(**********************SISSI:Swap from Ink to Storage Flush*********************************)
FUNCTION_BLOCK FB_Auto_Cycles_Swap
VAR_INPUT
	Sensor1			:BOOL;
	Sensor4			:BOOL;
	Circ_Pump_L	:BOOL;
	Circ_Pump_R	:BOOL;
	Circ_normal_error:INT;
	btPurge			:BOOL;
	
END_VAR
VAR_OUTPUT
	state								:INT;
	error_code					:INT;
	
	SwapInfo						:INT;
	VacValve_V8					:BOOL;	//白墨负压阀
	PurValve_V7					:BOOL;//正压阀
	alternate_Pumping		:BOOL;//交替加墨
	Swapping_Done			:BOOL;
	Error					:BOOL;
END_VAR
VAR
	step						:INT;
	stepA,stepB1,	stepB2		:INT;
	Ton,ton7,ton10				:TON;
	
	FB_SQUARE					:FB_SQUARE;
	W,X,A,Z,Y:INT;
	cycle_r_trig1,cycle_r_trig2  :R_TRIG;      //循坏
	cycle_x1,cycle_x2				:INT;//循坏次数
	purge_F_trig:F_TRIG;
	dely_off_setoff:TON;
	dely_emstop:Tc2_Standard.TON;
	ton1:Tc2_Standard.TON;
END_VAR
VAR_IN_OUT
	initialize				:BOOL;
	swap					:BOOL;
	CYCLE					:INT;//"0:Cycle A: Swap white ink to storage ;1:Cycle B: Swap storage to white ink"
	setoff					:BOOL;
END_VAR

IF setoff OR GVL.Reset THEN 
	step:=99;
END_IF
CASE step OF 
0://waiting
	IF initialize THEN 
		step :=5;
	ELSIF swap THEN 
		step :=10;
	ELSIF setoff OR GVL.Reset THEN 
		step :=99;
	END_IF
	
(***********当状态=Idle时，错误代码等于循坏错误****************************************)
	IF  state=MUStateEnum.idle THEN 
		error_code:=Circ_normal_error;
	END_IF
(***********自复位****************************************)	
	ton1(IN:=Swapping_Done , PT:= T#1S, Q=> , ET=> );
	IF ton1.Q THEN 
		Swapping_Done:=FALSE;
	END_IF
5://OFF
	state:=MUStateEnum.off;
	error_code:=MUErrorEnum.no_error;
	stepA:=stepB1:=stepB2:=0;
	W:=X:=A:=Z:=Y:=0;
	SwapInfo:=SwapInfoEnum.NONE;
	dely_emstop(IN:=FALSE);

	VacValve_V8:=FALSE;
	PurValve_V7:=FALSE;	
	
	GVL.fill_W_in_swap_enable:=FALSE;
	GVL.fill_F_in_swap_enable:=FALSE;
	
		IF initialize THEN //idle,此状态，所有泵停止	
			initialize:=FALSE;
			state:=MUStateEnum.idle;					
			GVL.fill_W_in_swap_enable:=FALSE;
			step:=0;
		END_IF
10://idle,此状态，所有泵停止				
		IF swap THEN 
			swap:=FALSE;
			state:=MUStateEnum.swapping;
			error_code:=MUErrorEnum.no_error;
			step:=20;
		END_IF
		
		IF error_code<>0 THEN 			
			step:=100;
		END_IF

20://SWAPPING		
		IF CYCLE=0 THEN
			ACT_Cycle_A();			
		ELSIF CYCLE=1 THEN 
			ACT_Cycle_B1();	
		END_IF
		
		IF SwapInfo=SwapInfoEnum.AC_STORAGE_FLUSH_FINISHED OR 
			SwapInfo=SwapInfoEnum.AC_WHITE_INK_FINISHED THEN 
			stepA:=stepB1:=stepB2:=0;		
			Swapping_Done:=TRUE;
			state:=MUStateEnum.idle;
			step:=0;
		END_IF
99://setoff
	setoff :=FALSE;
	error:=FALSE;
	state:=MUStateEnum.off;
	error_code:=MUErrorEnum.no_error;
	stepA:=stepB1:=stepB2:=0;
	W:=X:=A:=Z:=Y:=0;
	SwapInfo:=SwapInfoEnum.NONE;
	dely_emstop(IN:=FALSE);
	VacValve_V8:=FALSE;
	PurValve_V7:=FALSE;	
	
	GVL.fill_W_in_swap_enable:=FALSE;
	GVL.fill_F_in_swap_enable:=FALSE;
	step:=0;
100://error
		error:=TRUE;
		state:=MUStateEnum.error;
		stepA:=stepB1:=stepB2:=0;
		W:=X:=A:=Z:=Y:=0;
		dely_emstop(IN:=FALSE);
		VacValve_V8:=FALSE;
		PurValve_V7:=FALSE;	
		
		GVL.fill_W_in_swap_enable:=FALSE;
		GVL.fill_F_in_swap_enable:=FALSE;		
		step:=0;
END_CASE

IF setoff OR GVL.Reset THEN 
	step:=99;
END_IF

dely_off_setoff(IN:=setoff , PT:=T#1S , Q=> , ET=> );
IF dely_off_setoff.Q THEN
	setoff:=FALSE;
END_IF

IF state<>MUStateEnum.off AND state<>MUStateEnum.error  THEN 
	IF GVL.Emstop_Button THEN 
		error:=TRUE;
		error_code:=MUErrorEnum.emergency_error;
		PurValve_V7:=FALSE;
		dely_emstop(IN:=TRUE , PT:=T#1S , Q=> , ET=> );
		IF dely_emstop.Q THEN 
			VacValve_V8:=FALSE;
			step:=100;
		END_IF
	END_IF
END_IF

ACTION ACT_Cycle_A:
(***************Swap from White Ink to Storage Flush*******************************************)
CASE StepA OF
0:
	SwapInfo:=SwapInfoEnum.AC_STORAGE_FLUSH_RUNS;
	Ton(IN:=FALSE );	
	VacValve_V8:=FALSE;
	PurValve_V7 :=FALSE;
	stepA:=10;
10://SET "Vac White" OFF (valve 8 ON) 
	//START Pressure Purge Time = T1 (valve 7 ON)
	VacValve_V8:=TRUE;
	PurValve_V7 :=TRUE;
	Ton(IN:=TRUE , PT:=LREAL_TO_TIME(T[1]*1000) , Q=> , ET=> );
	IF Ton.Q THEN 
		Ton(IN:=FALSE );	
		stepA:=20;
	END_IF
20://STOP Pressure purge (normal filling conditions) (valve 7 OFF)	
	PurValve_V7:=FALSE;
	stepA:=30;
30://START Sol. filling (alternating pump time: T2=ON, T3=OFF)
	//WAIT UNTIL sensors in both TOP Sub Ink tanks detect a full tank (sensor 1 and 4)
	GVL.fill_F_in_swap_enable:=TRUE;
	alternate_Pumping:=TRUE;

	IF Sensor1 AND Sensor4 THEN 
		stepA:=31;
	END_IF
31://Wait Time: T4 (no vacuum)
	GVL.fill_F_in_swap_enable:=FALSE;
	alternate_Pumping:=FALSE;
	Ton(IN:=TRUE , PT:=LREAL_TO_TIME(T[4]*1000) , Q=> , ET=> );
		IF Ton.Q THEN 
			Ton(IN:=FALSE );
			stepA:=40;
		END_IF
40://Set "Vac White" ON  (Valve 8 OFF)     
	//Wait Time: T5 (filling conditions on & vac On)	
	VacValve_V8:=FALSE;	
	Ton(IN:=TRUE , PT:=LREAL_TO_TIME(T[5]*1000) , Q=> , ET=> );
	//调用加墨FB
		GVL.fill_F_in_swap_enable:=TRUE;
	IF Ton.Q THEN 
		stepA:=41;
	END_IF
41:
		GVL.fill_F_in_swap_enable:=FALSE;
		Ton(IN:=FALSE);
		stepA:=50;
50://Set "Vac White" Off (valve 8 ON)
	//For W=1 to 5 "Repeat 5x"
	//Pressure purge On for Time T6 (valve 7 ON)
	//Pressure purge Off for Time T6 (valve 7 OFF)
	VacValve_V8:=TRUE;
	FB_SQUARE(T_ON:=T[6] , T_OFF:=T[6] , SQUARE=>PurValve_V7 );
	purge_F_trig(CLK:=PurValve_V7 , Q=> );
	IF purge_F_trig.Q THEN 
		W:=W+1;
	END_IF
	
	IF W=6  THEN
		W:=0; 
		stepA:=60;
	END_IF
60://Wait  Time: T7 (while filling is ON)	
	Ton(IN:=TRUE  , PT:= LREAL_TO_TIME(T[7]*1000), Q=> , ET=> );	
	//调用加墨FB
	GVL.fill_F_in_swap_enable:=TRUE;
	IF ton.Q THEN 
		stepA:=61;
	END_IF
61:
		GVL.fill_F_in_swap_enable:=FALSE;
		Ton(IN:=FALSE);
		stepA:=70;
70://Set "Vac White" ON  (Valve 8 OFF)     
	//Wait Time: T5 (filling conditions on & vac On)
	VacValve_V8:=FALSE;
	//调用加墨FB
	GVL.fill_F_in_swap_enable:=TRUE;
	Ton(IN:=TRUE  , PT:= LREAL_TO_TIME(T[5]*1000), Q=> , ET=> );	
	IF ton.Q THEN 
		stepA:=71;
	END_IF
71:
		GVL.fill_F_in_swap_enable:=FALSE;
		Ton(IN:=FALSE);
		stepA:=80;
80://Set "Vac White" Off (valve 8 ON)
	VacValve_V8:=TRUE;
	//For X=1 to 5 "Repeat 5x"
	//Pressure purge On for Time T6 (valve 7 ON)
	//Pressure purge Off for Time T6 (valve 7 OFF)
	FB_SQUARE(T_ON:=T[6] , T_OFF:=T[6] , SQUARE=>PurValve_V7 );
	purge_F_trig(CLK:=PurValve_V7 , Q=> );
	IF purge_F_trig.Q THEN 
		X:=X+1;
	END_IF
	IF X=6  THEN 
		X:=0;
		stepA:=89;
	END_IF
89:
	A:=A+1;	
	stepA:=90;
90://Wait  Time: T7 (while filling is ON),第二次是T8	
	IF A<2 THEN 
		Ton(IN:=TRUE  , PT:= LREAL_TO_TIME(T[7]*1000), Q=> , ET=> );	
	ELSIF A=2 THEN 
		Ton(IN:=TRUE  , PT:= LREAL_TO_TIME(T[8]*1000), Q=> , ET=> );	
	END_IF
		//调用加墨FB
	GVL.fill_F_in_swap_enable:=TRUE;
	IF ton.Q THEN 
		stepA:=91;
	END_IF
91:
		GVL.fill_F_in_swap_enable:=FALSE;
		Ton(IN:=FALSE);
		stepA:=100;
100://Set "Vac White" ON  (Valve 8 OFF)    
	//Wait Time: T9 (filling conditions on) 
	VacValve_V8:=FALSE;
	//调用加墨FB
	GVL.fill_F_in_swap_enable:=TRUE;
	Ton(IN:=TRUE  , PT:= LREAL_TO_TIME(T[9]*1000), Q=> , ET=> );	
	IF ton.Q THEN 
		stepA:=101;
	END_IF	
101:
		GVL.fill_F_in_swap_enable:=FALSE;
		Ton(IN:=FALSE);
		stepA:=110;
110://重复	
	IF A<2 THEN 
		stepA:=10;
	ELSE stepA:=120;
	END_IF
120:(*FOR Z=1 to 5
	  IF both circulation pumps (3 & 6) were activated 3x within time: T13 => JUMP TO FINISH
	  ELSE Set Vac White Off (valve 8 ON)		
		NEXT Z*)
	A:=0;
	//	//调用加墨FB
	GVL.fill_F_in_swap_enable:=TRUE;
	Ton(IN:=TRUE  , PT:= LREAL_TO_TIME(T[13]*1000), Q=> , ET=> );	
	cycle_r_trig1(CLK:=Circ_Pump_L, Q=> );
	cycle_r_trig2(CLK:=Circ_Pump_R , Q=> );
		IF cycle_r_trig1.Q THEN 
			cycle_x1:=cycle_x1+1;
		END_IF
		IF cycle_r_trig2.Q THEN 
			cycle_x2:=cycle_x2+1;
		END_IF
		
	IF NOT Ton.Q AND cycle_x1>=3 AND cycle_x2>=3 THEN 
		Ton(IN:=FALSE);
		cycle_x1:=cycle_x2:=0;
		Z:=0;
		stepA:=190;
	ELSIF Ton.Q AND (cycle_x1<3 OR cycle_x2<3)  AND Z<5 THEN 	//循坏次数不够	
		Ton(IN:=FALSE);
		VacValve_V8:=TRUE;
		PurValve_V7:=TRUE;	
		cycle_x1:=cycle_x2:=0;
		stepA:=130;
	ELSIF Z=5 THEN
		Ton(IN:=FALSE);
		Z:=0; 
		stepA:=160;	
	END_IF
130://Start Pressure Purge On (valve 7 ON) for Time: T10
	//STOP Pressure purge (valve 7 OFF)   
			ton(IN:=TRUE , PT:= LREAL_TO_TIME(T[10]*1000) , Q=> , ET=> );		
			IF ton.Q THEN
				 ton(IN:=FALSE);
				PurValve_V7:=FALSE;
				stepA:=140;
			END_IF
140://Wait  Time: T7
		//Set "Vac White" ON  (Valve 8 OFF) 
			ton(IN:=TRUE , PT:= LREAL_TO_TIME(T[7]*1000) , Q=> , ET=> );
			IF Ton.Q THEN 
				ton(IN:=FALSE);
				VacValve_V8:=FALSE;		
				stepA:=150;
			END_IF
150://Wait Time: T11 (filling conditions on)
		//调用加墨FB
		ton(IN:=TRUE , PT:= LREAL_TO_TIME(T[11]*1000) , Q=> , ET=> );
			IF Ton.Q THEN 
				ton(IN:=FALSE);
				VacValve_V8:=FALSE;		
				Z:=Z+1;
				stepA:=120;
			END_IF
160://START WAIT = Message 2 on GUI 
	//If "PURGE BUTTON" is pushed during WAIT, THEN  
   //Set "Vac White" Off (valve 8 ON)
   //START Pressure purge (valve 7 ON) until button released
		SwapInfo:=SwapInfoEnum.AC_STORAGE_FLUSH_NEEDS_HELP;
			VacValve_V8:=TRUE;
		IF btPurge THEN 			
			PurValve_V7:=TRUE;
			stepA:=170;
		END_IF
170:    //START Pressure purge (valve 7 ON) until button released
		IF NOT btPurge THEN 
			PurValve_V7:=FALSE;
			stepA:=171;
		END_IF
171://Wait  Time: T7
	//Set "Vac White" ON  (Valve 8 OFF)  
		ton(IN:=TRUE , PT:= LREAL_TO_TIME(T[7]*1000) , Q=> , ET=> );
			IF Ton.Q THEN 
				ton(IN:=FALSE);
				VacValve_V8:=FALSE;
				stepA:=180;
			END_IF
180://  IF both circulation pumps (3 & 6) were activated 3x within time: T13 => JUMP TO FINISH
			//END IF (back TO wait)
		//	//调用加墨FB
	Ton(IN:=TRUE  , PT:= LREAL_TO_TIME(T[13]*1000), Q=> , ET=> );	
	cycle_r_trig1(CLK:=Circ_Pump_L, Q=> );
	cycle_r_trig2(CLK:=Circ_Pump_R , Q=> );
		IF cycle_r_trig1.Q THEN 
			cycle_x1:=cycle_x1+1;
		END_IF
		IF cycle_r_trig2.Q THEN 
			cycle_x2:=cycle_x2+1;
		END_IF
	IF NOT Ton.Q AND cycle_x1>=3 AND cycle_x2>=3 THEN 
		Ton(IN:=FALSE);
		cycle_x1:=cycle_x2:=0;
		stepA:=190;
	ELSIF Ton.Q AND (cycle_x1<3 OR cycle_x2<3) THEN 		
		Ton(IN:=FALSE);
		cycle_x1:=cycle_x2:=0;
		stepA:=160;
	END_IF
190:	//关闭所有供墨
	GVL.fill_F_in_swap_enable:=FALSE;
	stepA:=200;
200://FINISH => Message 3 on GUI
		SwapInfo:=SwapInfoEnum.AC_STORAGE_FLUSH_FINISHED;
		
END_CASE
END_ACTION

ACTION ACT_Cycle_B1:
(*************** Swap From Storage Flush to White Ink*******************************************)
CASE StepB1 OF
0:
	SwapInfo:=SwapInfoEnum.AC_WHITE_INK_RUNS;
	Ton(IN:=FALSE );	
	VacValve_V8:=FALSE;
	PurValve_V7 :=FALSE;
	StepB1:=10;
10://SET "Vac White" OFF (valve 8 ON) 
	//START Pressure Purge Time = T1 (valve 7 ON)
	VacValve_V8:=TRUE;
	PurValve_V7 :=TRUE;
	Ton(IN:=TRUE , PT:=LREAL_TO_TIME(T[1]*1000) , Q=> , ET=> );
	IF Ton.Q THEN 
		Ton(IN:=FALSE );	
		StepB1:=20;
	END_IF
20://STOP Pressure purge (normal filling conditions) (valve 7 OFF)	
	PurValve_V7:=FALSE;
	StepB1:=30;
30://START Ink filling  (alternating pump time: T2=ON, T3=OFF)
	//WAIT UNTIL sensors in both TOP Sub Ink tanks detect a full tank (sensor 1 and 4)	
	GVL.fill_W_in_swap_enable:=TRUE;
	alternate_Pumping:=TRUE;
	
	IF Sensor1 AND Sensor4 THEN 
		StepB1:=31;
	END_IF
31://Wait Time: T4 (no vacuum)
	GVL.fill_W_in_swap_enable:=FALSE;
	alternate_Pumping:=FALSE;
	Ton(IN:=TRUE , PT:=LREAL_TO_TIME(T[4]*1000) , Q=> , ET=> );
		IF Ton.Q THEN 
			Ton(IN:=FALSE );
			StepB1:=40;
		END_IF
40://Set "Vac White" ON  (Valve 8 OFF)     
	//Wait Time: T5 (filling conditions on & vac On)	
	VacValve_V8:=FALSE;	
	Ton(IN:=TRUE , PT:=LREAL_TO_TIME(T[5]*1000) , Q=> , ET=> );
	//调用加墨FB
		GVL.fill_W_in_swap_enable:=TRUE;
	IF Ton.Q THEN 
		StepB1:=41;
	END_IF
41:
		GVL.fill_W_in_swap_enable:=FALSE;
		Ton(IN:=FALSE);
		StepB1:=50;
50://Set "Vac White" Off (valve 8 ON)
	//For Z=1 to 5 "Repeat 5x"
	//Pressure purge On for Time T6 (valve 7 ON)
	//Pressure purge Off for Time T6 (valve 7 OFF)
	VacValve_V8:=TRUE;
	FB_SQUARE(T_ON:=T[6] , T_OFF:=T[6] , SQUARE=>PurValve_V7 );
	purge_F_trig(CLK:=PurValve_V7 , Q=> );
	IF purge_F_trig.Q THEN 
		Z:=Z+1;
	END_IF
	
	IF Z=6  THEN
		Z:=0; 
		StepB1:=60;
	END_IF
60://Wait  Time: T7
	Ton(IN:=TRUE  , PT:= LREAL_TO_TIME(T[7]*1000), Q=> , ET=> );	
	//调用加墨FB
	GVL.fill_W_in_swap_enable:=TRUE;
	IF ton.Q THEN 
		StepB1:=61;
	END_IF
61:
		GVL.fill_W_in_swap_enable:=FALSE;
		Ton(IN:=FALSE);
		StepB1:=70;
70://Set "Vac White" ON  (Valve 8 OFF)     
	//Wait Time: T5 (filling conditions on & vac On)
	VacValve_V8:=FALSE;
	//调用加墨FB
	GVL.fill_W_in_swap_enable:=TRUE;
	Ton(IN:=TRUE  , PT:= LREAL_TO_TIME(T[5]*1000), Q=> , ET=> );	
	IF ton.Q THEN 
		StepB1:=71;
	END_IF
71:
		GVL.fill_W_in_swap_enable:=FALSE;
		Ton(IN:=FALSE);
		StepB1:=80;
80://Set "Vac White" Off (valve 8 ON)
	VacValve_V8:=TRUE;
	//For Z=1 to 5 "Repeat 5x"
	//Pressure purge On for Time T6 (valve 7 ON)
	//Pressure purge Off for Time T6 (valve 7 OFF)
	FB_SQUARE(T_ON:=T[6] , T_OFF:=T[6] , SQUARE=>PurValve_V7 );
	purge_F_trig(CLK:=PurValve_V7 , Q=> );
	IF purge_F_trig.Q THEN 
		Z:=Z+1;
	END_IF
	IF Z=6  THEN 
		Z:=0;
		StepB1:=90;
	END_IF
90://Wait Time: T8 (filling conditions on, vac off))
		Ton(IN:=TRUE  , PT:= LREAL_TO_TIME(T[8]*1000), Q=> , ET=> );	
		//调用加墨FB
	GVL.fill_W_in_swap_enable:=TRUE;
	IF ton.Q THEN 
		StepB1:=91;
	END_IF
91:
		GVL.fill_W_in_swap_enable:=FALSE;
		Ton(IN:=FALSE);
		StepB1:=100;
100://Set "Vac White" ON  (Valve 8 OFF)    
	//Wait Time: T9 (filling conditions on) 
	VacValve_V8:=FALSE;
	//调用加墨FB
	GVL.fill_W_in_swap_enable:=TRUE;
	Ton(IN:=TRUE  , PT:= LREAL_TO_TIME(T[9]*1000), Q=> , ET=> );	
	IF ton.Q THEN 
		StepB1:=101;
	END_IF	
101:
		GVL.fill_W_in_swap_enable:=FALSE;
		Ton(IN:=FALSE);
		StepB1:=110;
110://无重复
		StepB1:=120;
120:(*FOR Y=1 to 5
	  IF both circulation pumps (3 & 6) were activated 3x within time: T13 => JUMP TO PAUSE
	  ELSE Set Vac White Off (valve 8 ON)		
		NEXT Y*)
	//	//调用加墨FB
	GVL.fill_W_in_swap_enable:=TRUE;
	Ton(IN:=TRUE  , PT:= LREAL_TO_TIME(T[13]*1000), Q=> , ET=> );	
	cycle_r_trig1(CLK:=Circ_Pump_L, Q=> );
	cycle_r_trig2(CLK:=Circ_Pump_R , Q=> );
		IF cycle_r_trig1.Q THEN 
			cycle_x1:=cycle_x1+1;
		END_IF
		IF cycle_r_trig2.Q THEN 
			cycle_x2:=cycle_x2+1;
		END_IF
		
	IF NOT Ton.Q AND cycle_x1>=3 AND cycle_x2>=3 THEN 
		Ton(IN:=FALSE);
		cycle_x1:=cycle_x2:=0;
		Y:=0;
		StepB1:=200;
	ELSIF Ton.Q AND (cycle_x1<3 OR cycle_x2<3)  AND Z<5 THEN 	//循坏次数不够,ELSE Set Vac White Off (valve 8 ON	
		Ton(IN:=FALSE);
		VacValve_V8:=TRUE;
		PurValve_V7:=TRUE;	
		cycle_x1:=cycle_x2:=0;
		StepB1:=130;
	ELSIF Y=5 THEN
		Ton(IN:=FALSE);
		Y:=0; 
		StepB1:=160;	
	END_IF
130://Start Pressure Purge On (valve 7 ON) for Time: T10
	//STOP Pressure purge (valve 7 OFF)   
			ton(IN:=TRUE , PT:= LREAL_TO_TIME(T[10]*1000) , Q=> , ET=> );		
			IF ton.Q THEN
				 ton(IN:=FALSE);
				PurValve_V7:=FALSE;
				StepB1:=140;
			END_IF
140://Wait  Time: T7
		//Set "Vac White" ON  (Valve 8 OFF) 
			ton(IN:=TRUE , PT:= LREAL_TO_TIME(T[7]*1000) , Q=> , ET=> );
			IF Ton.Q THEN 
				ton(IN:=FALSE);
				VacValve_V8:=FALSE;		
				StepB1:=150;
			END_IF
150://Wait Time: T11 (filling conditions on)
		//调用加墨FB
		ton(IN:=TRUE , PT:= LREAL_TO_TIME(T[11]*1000) , Q=> , ET=> );
			IF Ton.Q THEN 
				ton(IN:=FALSE);
				VacValve_V8:=FALSE;		
				Y:=Y+1;
				StepB1:=120;
			END_IF
160://START WAIT = Message 5 on GUI 
	//If "PURGE BUTTON" is pushed during WAIT, THEN  
   //Set "Vac White" Off (valve 8 ON)
   //START Pressure purge (valve 7 ON) until button released
		SwapInfo:=SwapInfoEnum.AC_WHITE_INK1_NEEDS_HELP;
			VacValve_V8:=TRUE;
		IF btPurge THEN 		
			PurValve_V7:=TRUE;
			StepB1:=170;
		END_IF
170:    //START Pressure purge (valve 7 ON) until button released
		IF NOT btPurge THEN 
			PurValve_V7:=FALSE;
			StepB1:=171;
		END_IF
171://Wait  Time: T7
	//Set "Vac White" ON  (Valve 8 OFF)  
		ton(IN:=TRUE , PT:= LREAL_TO_TIME(T[7]*1000) , Q=> , ET=> );
			IF Ton.Q THEN 
				ton(IN:=FALSE);
				VacValve_V8:=FALSE;
				StepB1:=180;
			END_IF
180://  IF both circulation pumps (3 & 6) were activated 3x within time T13 than:
		//           => remove Message 5
		//           => Show Message 4
		//           => JUMP TO PAUSE
		//END IF (back to wait)
				
		//	//调用加墨FB
	Ton(IN:=TRUE  , PT:= LREAL_TO_TIME(T[13]*1000), Q=> , ET=> );	
	cycle_r_trig1(CLK:=Circ_Pump_L, Q=> );
	cycle_r_trig2(CLK:=Circ_Pump_R , Q=> );
		IF cycle_r_trig1.Q THEN 
			cycle_x1:=cycle_x1+1;
		END_IF
		IF cycle_r_trig2.Q THEN 
			cycle_x2:=cycle_x2+1;
		END_IF
	IF NOT Ton.Q AND cycle_x1>=3 AND cycle_x2>=3 THEN 
		Ton(IN:=FALSE);
		cycle_x1:=cycle_x2:=0;
		StepB1:=190;
	ELSIF Ton.Q AND (cycle_x1<3 OR cycle_x2<3) THEN 		
		Ton(IN:=FALSE);
		cycle_x1:=cycle_x2:=0;
		StepB1:=160;
	END_IF
190:	//           => remove Message 5
		//           => Show Message 4
		//           => JUMP TO PAUSE
	SwapInfo:=SwapInfoEnum.AC_WHITE_INK_RUNS;	
	GVL.fill_W_in_swap_enable:=FALSE;
	StepB1:=200;
200://PAUSE:  wait time time: T12,Filter cleaning time
	//调用加墨FB
	GVL.fill_W_in_swap_enable:=TRUE;
	Ton(IN:=TRUE  , PT:= LREAL_TO_TIME(T[12]*1000), Q=> , ET=> );	
	IF Ton.Q THEN 
		StepB1:=210;		
	END_IF
210://关闭加墨
		Ton(IN:=FALSE);
		GVL.fill_W_in_swap_enable:=FALSE;
		StepB1:=220;
220://
	ACT_Cycle_B2();
		
END_CASE
END_ACTION

ACTION ACT_Cycle_B2:
(*************** Swap From Storage Flush to White Ink*******************************************)

CASE StepB2 OF
0:
	Ton(IN:=FALSE );	
	StepB2:=10;
10://SET "Vac White" OFF (valve 8 ON) 
	//START Pressure Purge Time = T1 (valve 7 ON)
	VacValve_V8:=TRUE;
	PurValve_V7 :=TRUE;
	Ton(IN:=TRUE , PT:=LREAL_TO_TIME(T[1]*1000) , Q=> , ET=> );
	IF Ton.Q THEN 
		Ton(IN:=FALSE );	
		StepB2:=20;
	END_IF
20://STOP Pressure purge (normal filling conditions) (valve 7 OFF)	
	PurValve_V7:=FALSE;
	StepB2:=30;
30://START Ink filling  (alternating pump time: T2=ON, T3=OFF)
	//WAIT UNTIL sensors in both TOP Sub Ink tanks detect a full tank (sensor 1 and 4)
	GVL.fill_W_in_swap_enable:=TRUE;
	alternate_Pumping:=TRUE;
	
	IF Sensor1 AND Sensor4 THEN 
		StepB2:=31;
	END_IF
31://Wait Time: T4 (no vacuum)
	GVL.fill_W_in_swap_enable:=FALSE;
	alternate_Pumping:=FALSE;
	Ton(IN:=TRUE , PT:=LREAL_TO_TIME(T[4]*1000) , Q=> , ET=> );
		IF Ton.Q THEN 
			Ton(IN:=FALSE );
			StepB2:=40;
		END_IF
40://Set "Vac White" ON  (Valve 8 OFF)     
	//Wait Time: T5 (filling conditions on & vac On)	
	VacValve_V8:=FALSE;	
	Ton(IN:=TRUE , PT:=LREAL_TO_TIME(T[5]*1000) , Q=> , ET=> );
	//调用加墨FB
		GVL.fill_W_in_swap_enable:=TRUE;
	IF Ton.Q THEN 
		StepB2:=41;
	END_IF
41:
		GVL.fill_W_in_swap_enable:=FALSE;
		Ton(IN:=FALSE);
		StepB2:=50;
50://Set "Vac White" Off (valve 8 ON)
	//For Z=1 to 5 "Repeat 5x"
	//Pressure purge On for Time T6 (valve 7 ON)
	//Pressure purge Off for Time T6 (valve 7 OFF)
	VacValve_V8:=TRUE;
	FB_SQUARE(T_ON:=T[6] , T_OFF:=T[6] , SQUARE=>PurValve_V7 );
	purge_F_trig(CLK:=PurValve_V7 , Q=> );
	IF purge_F_trig.Q THEN 
		Z:=Z+1;
	END_IF
	
	IF Z=6  THEN
		Z:=0; 
		StepB2:=60;
	END_IF
60://Wait  Time: T7
	Ton(IN:=TRUE  , PT:= LREAL_TO_TIME(T[7]*1000), Q=> , ET=> );	
	//调用加墨FB
	GVL.fill_W_in_swap_enable:=TRUE;
	IF ton.Q THEN 
		StepB2:=61;
	END_IF
61:
		GVL.fill_W_in_swap_enable:=FALSE;
		Ton(IN:=FALSE);
		StepB2:=70;
70://Set "Vac White" ON  (Valve 8 OFF)     
	//Wait Time: T5 (filling conditions on & vac On)
	VacValve_V8:=FALSE;
	//调用加墨FB
	GVL.fill_W_in_swap_enable:=TRUE;
	Ton(IN:=TRUE  , PT:= LREAL_TO_TIME(T[5]*1000), Q=> , ET=> );	
	IF ton.Q THEN 
		StepB2:=71;
	END_IF
71:
		GVL.fill_W_in_swap_enable:=FALSE;
		Ton(IN:=FALSE);
		StepB2:=80;
80://Set "Vac White" Off (valve 8 ON)
	VacValve_V8:=TRUE;
	//For Z=1 to 5 "Repeat 5x"
	//Pressure purge On for Time T6 (valve 7 ON)
	//Pressure purge Off for Time T6 (valve 7 OFF)
	FB_SQUARE(T_ON:=T[6] , T_OFF:=T[6] , SQUARE=>PurValve_V7 );
	purge_F_trig(CLK:=PurValve_V7 , Q=> );
	IF purge_F_trig.Q THEN 
		Z:=Z+1;
	END_IF
	IF Z=6  THEN 
		Z:=0;
		StepB2:=90;
	END_IF
90://Wait Time: T8 (filling conditions on, vac off))
		Ton(IN:=TRUE  , PT:= LREAL_TO_TIME(T[8]*1000), Q=> , ET=> );	
		//调用加墨FB
	GVL.fill_W_in_swap_enable:=TRUE;
	IF ton.Q THEN 
		StepB2:=91;
	END_IF
91:
		GVL.fill_W_in_swap_enable:=FALSE;
		Ton(IN:=FALSE);
		StepB2:=100;
100://Set "Vac White" ON  (Valve 8 OFF)    
	//Wait Time: T9 (filling conditions on) 
	VacValve_V8:=FALSE;
	//调用加墨FB
	GVL.fill_W_in_swap_enable:=TRUE;
	Ton(IN:=TRUE  , PT:= LREAL_TO_TIME(T[9]*1000), Q=> , ET=> );	
	IF ton.Q THEN 
		StepB2:=101;
	END_IF	
101:
		GVL.fill_W_in_swap_enable:=FALSE;
		Ton(IN:=FALSE);
		StepB2:=110;
110://无重复
		StepB2:=120;
120:(*FOR Z=1 to 5
	  IF both circulation pumps (3 & 6) were activated 3x within time: T13 => JUMP TO FINISH
	  ELSE Set Vac White Off (valve 8 ON)		
		NEXT Z*)
	//	//调用加墨FB
	GVL.fill_W_in_swap_enable:=TRUE;
	Ton(IN:=TRUE  , PT:= LREAL_TO_TIME(T[13]*1000), Q=> , ET=> );	
	cycle_r_trig1(CLK:=Circ_Pump_L, Q=> );
	cycle_r_trig2(CLK:=Circ_Pump_R , Q=> );
		IF cycle_r_trig1.Q THEN 
			cycle_x1:=cycle_x1+1;
		END_IF
		IF cycle_r_trig2.Q THEN 
			cycle_x2:=cycle_x2+1;
		END_IF
		
	IF NOT Ton.Q AND cycle_x1>=3 AND cycle_x2>=3 THEN 
		Ton(IN:=FALSE);
		cycle_x1:=cycle_x2:=0;
		Z:=0;
		StepB2:=200;
	ELSIF Ton.Q AND (cycle_x1<3 OR cycle_x2<3)  AND Z<5 THEN 	//循坏次数不够,ELSE Set Vac White Off (valve 8 ON	
		Ton(IN:=FALSE);
		VacValve_V8:=TRUE;
		PurValve_V7:=TRUE;	
		cycle_x1:=cycle_x2:=0;
		StepB2:=130;
	ELSIF Z=5 THEN
		Ton(IN:=FALSE);
		Z:=0; 
		StepB2:=160;	
	END_IF
130://Start Pressure Purge On (valve 7 ON) for Time: T10
	//STOP Pressure purge (valve 7 OFF)   
			ton(IN:=TRUE , PT:= LREAL_TO_TIME(T[10]*1000) , Q=> , ET=> );		
			IF ton.Q THEN
				 ton(IN:=FALSE);
				PurValve_V7:=FALSE;
				StepB2:=140;
			END_IF
140://Wait  Time: T7
		//Set "Vac White" ON  (Valve 8 OFF) 
			ton(IN:=TRUE , PT:= LREAL_TO_TIME(T[7]*1000) , Q=> , ET=> );
			IF Ton.Q THEN 
				ton(IN:=FALSE);
				VacValve_V8:=FALSE;		
				StepB2:=150;
			END_IF
150://Wait Time: T11 (filling conditions on)
		//调用加墨FB
		ton(IN:=TRUE , PT:= LREAL_TO_TIME(T[11]*1000) , Q=> , ET=> );
			IF Ton.Q THEN 
				ton(IN:=FALSE);
				VacValve_V8:=FALSE;		
				Z:=Z+1;
				StepB2:=120;
			END_IF
160://START WAIT = Message 6 on GUI 
	//If "PURGE BUTTON" is pushed during WAIT, THEN  
   //Set "Vac White" Off (valve 8 ON)
   //START Pressure purge (valve 7 ON) until button released
		SwapInfo:=SwapInfoEnum.AC_WHITE_INK2_NEEDS_HELP;
			VacValve_V8:=TRUE;
		IF btPurge THEN 			
			PurValve_V7:=TRUE;
			StepB2:=170;
		END_IF
170:    //START Pressure purge (valve 7 ON) until button released
		IF NOT btPurge THEN 
			PurValve_V7:=FALSE;
			StepB2:=171;
		END_IF
171://Wait  Time: T7
	//Set "Vac White" ON  (Valve 8 OFF)  
		ton(IN:=TRUE , PT:= LREAL_TO_TIME(T[7]*1000) , Q=> , ET=> );
			IF Ton.Q THEN 
				ton(IN:=FALSE);
				VacValve_V8:=FALSE;
				StepB2:=180;
			END_IF
180://    IF both circulation pumps (3 & 6) were activated 3x within time: T13 => JUMP TO FINISH
		//END IF (back to wait)
				
		//	//调用加墨FB
	Ton(IN:=TRUE  , PT:= LREAL_TO_TIME(T[13]*1000), Q=> , ET=> );	
	cycle_r_trig1(CLK:=Circ_Pump_L, Q=> );
	cycle_r_trig2(CLK:=Circ_Pump_R , Q=> );
		IF cycle_r_trig1.Q THEN 
			cycle_x1:=cycle_x1+1;
		END_IF
		IF cycle_r_trig2.Q THEN 
			cycle_x2:=cycle_x2+1;
		END_IF
	IF NOT Ton.Q AND cycle_x1>=3 AND cycle_x2>=3 THEN 
		Ton(IN:=FALSE);
		cycle_x1:=cycle_x2:=0;
		StepB2:=190;
	ELSIF Ton.Q AND (cycle_x1<3 OR cycle_x2<3) THEN 		
		Ton(IN:=FALSE);
		cycle_x1:=cycle_x2:=0;
		StepB2:=160;
	END_IF
190:	//  
	StepB2:=200;
200://
	StepB2:=210;
210://关闭加墨
	Ton(IN:=FALSE);
	GVL.fill_W_in_swap_enable:=FALSE;
	StepB2:=220;
220://FINISH => Message 7 on GUI
	SwapInfo:=SwapInfoEnum.AC_WHITE_INK_FINISHED;

		
END_CASE
END_ACTION

END_FUNCTION_BLOCK

(* stored: Version 1.1.0.1, ProductVersion 3.1.4024.11
   POU FB_Auto_Cycles_Swap: Id {6179c9e0-e6d3-4e26-93a6-fb67a88fabce}, SpecialFunc None
   Action ACT_Cycle_A: Id {184a14f9-54ea-4235-99d8-0e356b46053a}
   Action ACT_Cycle_B1: Id {59399709-08cf-4668-b4ea-c4ca4657029e}
   Action ACT_Cycle_B2: Id {de859a24-cb09-4428-a859-6ce7c323b729} *)
